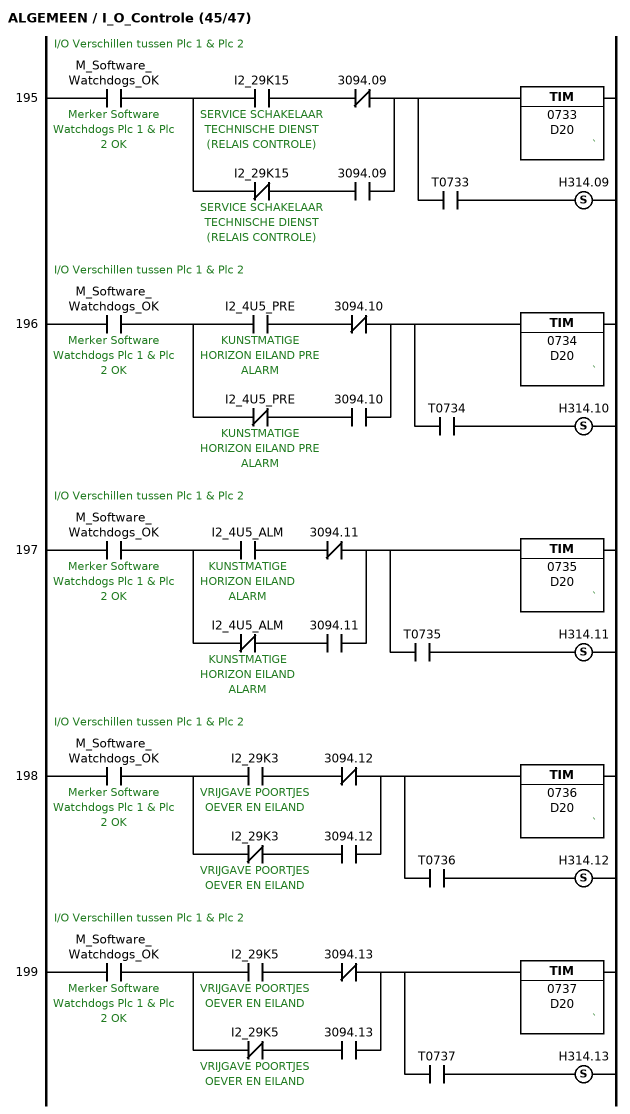
; [picture p253: ALGEMEEN / I_O_Controle, rungs 195-199]
; rung 195: I/O Verschillen tussen Plc 1 & Plc 2
LD M_Software_Watchdogs_OK  ; Merker Software Watchdogs Plc 1 & Plc 2 OK
LD I2_29K15  ; SERVICE SCHAKELAAR TECHNISCHE DIENST (RELAIS CONTROLE)
ANDNOT 3094.09
LDNOT I2_29K15  ; SERVICE SCHAKELAAR TECHNISCHE DIENST (RELAIS CONTROLE)
AND 3094.09
ORLD
ANDLD
TIM 0733 D20  ; `
AND T0733
SET H314.09
; rung 196: I/O Verschillen tussen Plc 1 & Plc 2
LD M_Software_Watchdogs_OK  ; Merker Software Watchdogs Plc 1 & Plc 2 OK
LD I2_4U5_PRE  ; KUNSTMATIGE HORIZON EILAND PRE ALARM
ANDNOT 3094.10
LDNOT I2_4U5_PRE  ; KUNSTMATIGE HORIZON EILAND PRE ALARM
AND 3094.10
ORLD
ANDLD
TIM 0734 D20  ; `
AND T0734
SET H314.10
; rung 197: I/O Verschillen tussen Plc 1 & Plc 2
LD M_Software_Watchdogs_OK  ; Merker Software Watchdogs Plc 1 & Plc 2 OK
LD I2_4U5_ALM  ; KUNSTMATIGE HORIZON EILAND ALARM
ANDNOT 3094.11
LDNOT I2_4U5_ALM  ; KUNSTMATIGE HORIZON EILAND ALARM
AND 3094.11
ORLD
ANDLD
TIM 0735 D20  ; `
AND T0735
SET H314.11
; rung 198: I/O Verschillen tussen Plc 1 & Plc 2
LD M_Software_Watchdogs_OK  ; Merker Software Watchdogs Plc 1 & Plc 2 OK
LD I2_29K3  ; VRIJGAVE POORTJES OEVER EN EILAND
ANDNOT 3094.12
LDNOT I2_29K3  ; VRIJGAVE POORTJES OEVER EN EILAND
AND 3094.12
ORLD
ANDLD
TIM 0736 D20  ; `
AND T0736
SET H314.12
; rung 199: I/O Verschillen tussen Plc 1 & Plc 2
LD M_Software_Watchdogs_OK  ; Merker Software Watchdogs Plc 1 & Plc 2 OK
LD I2_29K5  ; VRIJGAVE POORTJES OEVER EN EILAND
ANDNOT 3094.13
LDNOT I2_29K5  ; VRIJGAVE POORTJES OEVER EN EILAND
AND 3094.13
ORLD
ANDLD
TIM 0737 D20  ; `
AND T0737
SET H314.13

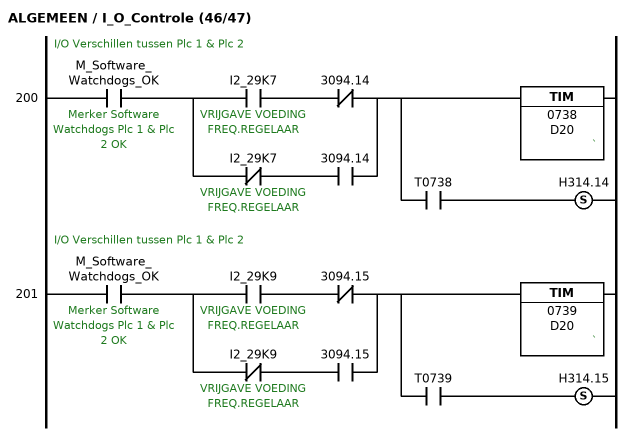
; rung 200: I/O Verschillen tussen Plc 1 & Plc 2
LD M_Software_Watchdogs_OK  ; Merker Software Watchdogs Plc 1 & Plc 2 OK
LD I2_29K7  ; VRIJGAVE VOEDING FREQ.REGELAAR
ANDNOT 3094.14
LDNOT I2_29K7  ; VRIJGAVE VOEDING FREQ.REGELAAR
AND 3094.14
ORLD
ANDLD
TIM 0738 D20  ; `
AND T0738
SET H314.14
; rung 201: I/O Verschillen tussen Plc 1 & Plc 2
LD M_Software_Watchdogs_OK  ; Merker Software Watchdogs Plc 1 & Plc 2 OK
LD I2_29K9  ; VRIJGAVE VOEDING FREQ.REGELAAR
ANDNOT 3094.15
LDNOT I2_29K9  ; VRIJGAVE VOEDING FREQ.REGELAAR
AND 3094.15
ORLD
ANDLD
TIM 0739 D20  ; `
AND T0739
SET H314.15

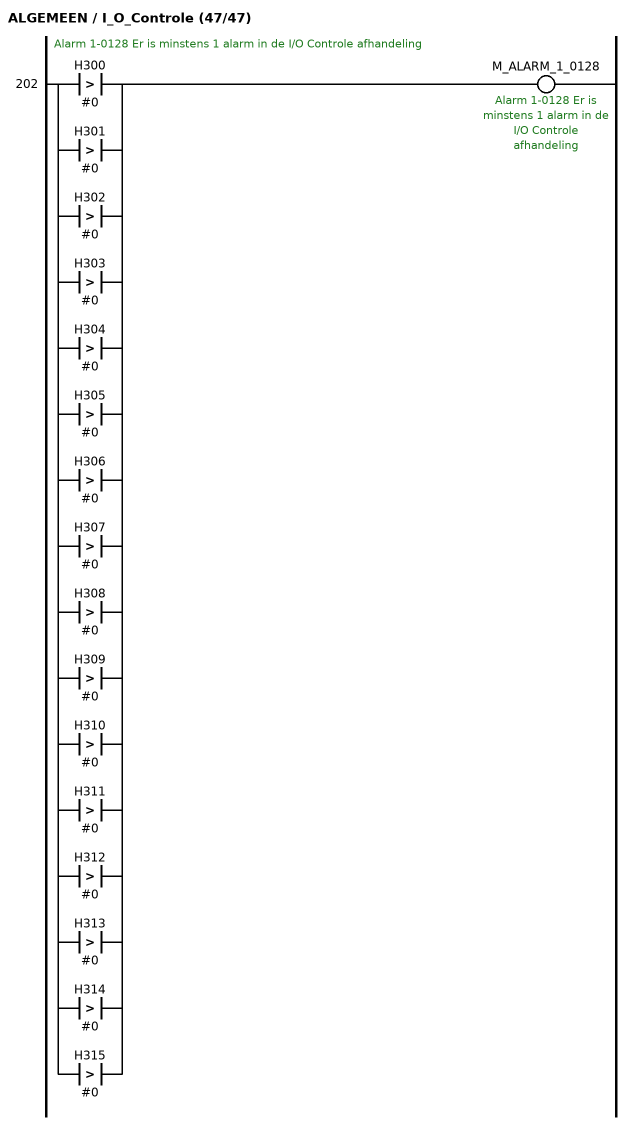
; rung 202: Alarm 1-0128 Er is minstens 1 alarm in de I/O Controle afhandeling
LD>(320) H300 #0
OR>(320) H301 #0
OR>(320) H302 #0
OR>(320) H303 #0
OR>(320) H304 #0
OR>(320) H305 #0
OR>(320) H306 #0
OR>(320) H307 #0
OR>(320) H308 #0
OR>(320) H309 #0
OR>(320) H310 #0
OR>(320) H311 #0
OR>(320) H312 #0
OR>(320) H313 #0
OR>(320) H314 #0
OR>(320) H315 #0
OUT M_ALARM_1_0128  ; Alarm 1-0128 Er is minstens 1 alarm in de I/O Controle afhandeling

### Section Voedingen

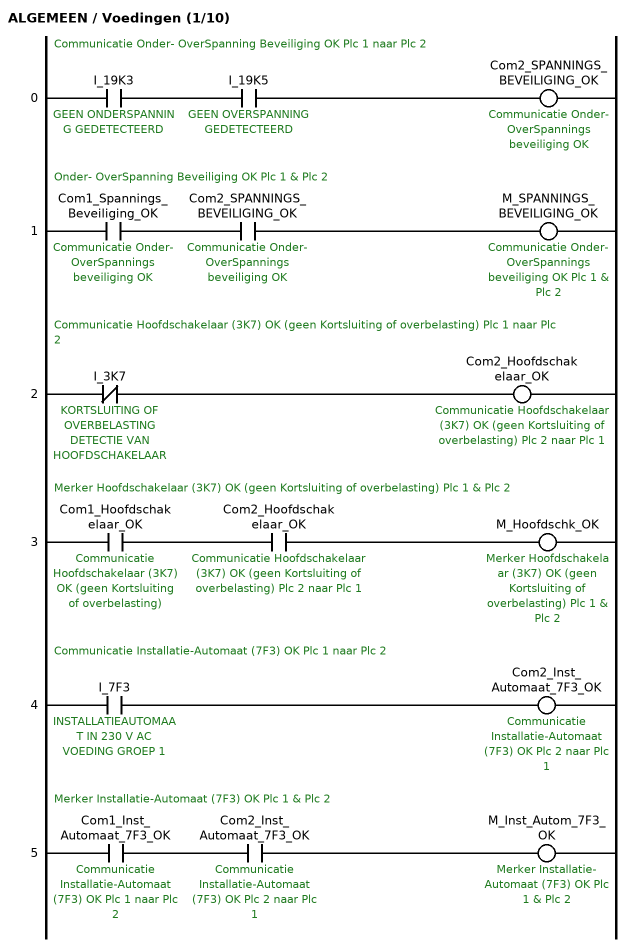
; rung 0: Communicatie Onder- OverSpanning Beveiliging OK Plc 1 naar Plc 2
LD I_19K3  ; GEEN ONDERSPANNING GEDETECTEERD
AND I_19K5  ; GEEN OVERSPANNING GEDETECTEERD
OUT Com2_SPANNINGS_BEVEILIGING_OK  ; Communicatie Onder- OverSpannings beveiliging OK
; rung 1: Onder- OverSpanning Beveiliging OK Plc 1 & Plc 2
LD Com1_Spannings_Beveiliging_OK  ; Communicatie Onder- OverSpannings beveiliging OK
AND Com2_SPANNINGS_BEVEILIGING_OK  ; Communicatie Onder- OverSpannings beveiliging OK
OUT M_SPANNINGS_BEVEILIGING_OK  ; Communicatie Onder- OverSpannings beveiliging OK Plc 1 & Plc 2
; rung 2: Communicatie Hoofdschakelaar (3K7) OK (geen Kortsluiting of overbelasting) Plc 1 naar Plc 2
LDNOT I_3K7  ; KORTSLUITING OF OVERBELASTING DETECTIE VAN HOOFDSCHAKELAAR
OUT Com2_Hoofdschakelaar_OK  ; Communicatie Hoofdschakelaar (3K7) OK (geen Kortsluiting of overbelasting) Plc 2 naar Plc 1
; rung 3: Merker Hoofdschakelaar (3K7) OK (geen Kortsluiting of overbelasting) Plc 1 & Plc 2
LD Com1_Hoofdschakelaar_OK  ; Communicatie Hoofdschakelaar (3K7) OK (geen Kortsluiting of overbelasting)
AND Com2_Hoofdschakelaar_OK  ; Communicatie Hoofdschakelaar (3K7) OK (geen Kortsluiting of overbelasting) Plc 2 naar Plc 1
OUT M_Hoofdschk_OK  ; Merker Hoofdschakelaar (3K7) OK (geen Kortsluiting of overbelasting) Plc 1 & Plc 2
; rung 4: Communicatie Installatie-Automaat (7F3) OK Plc 1 naar Plc 2
LD I_7F3  ; INSTALLATIEAUTOMAAT IN 230 V AC VOEDING GROEP 1
OUT Com2_Inst_Automaat_7F3_OK  ; Communicatie Installatie-Automaat (7F3) OK Plc 2 naar Plc 1
; rung 5: Merker Installatie-Automaat (7F3) OK Plc 1 & Plc 2
LD Com1_Inst_Automaat_7F3_OK  ; Communicatie Installatie-Automaat (7F3) OK Plc 1 naar Plc 2
AND Com2_Inst_Automaat_7F3_OK  ; Communicatie Installatie-Automaat (7F3) OK Plc 2 naar Plc 1
OUT M_Inst_Autom_7F3_OK  ; Merker Installatie-Automaat (7F3) OK Plc 1 & Plc 2

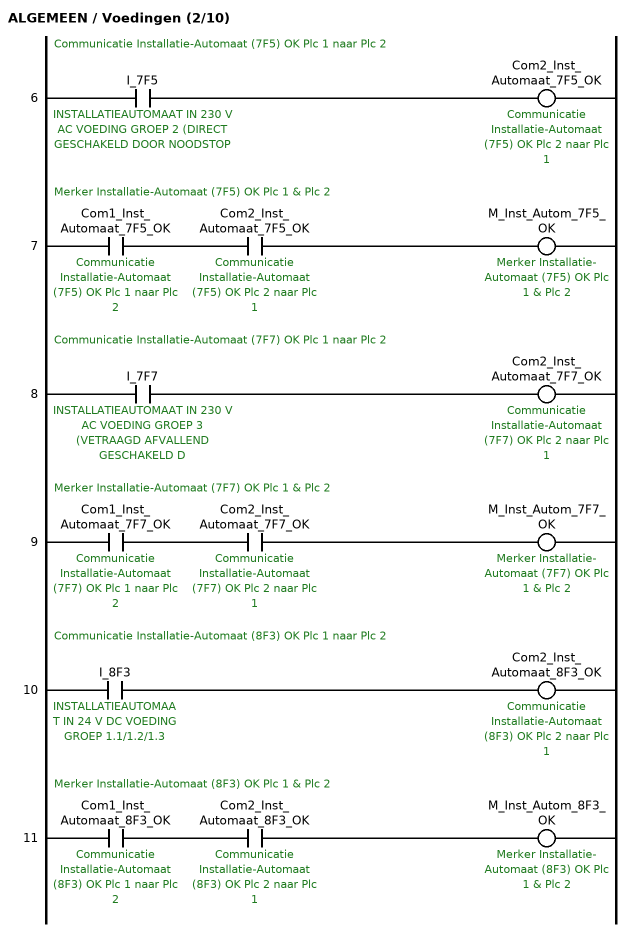
; rung 6: Communicatie Installatie-Automaat (7F5) OK Plc 1 naar Plc 2
LD I_7F5  ; INSTALLATIEAUTOMAAT IN 230 V AC VOEDING GROEP 2 (DIRECT GESCHAKELD DOOR NOODSTOP
OUT Com2_Inst_Automaat_7F5_OK  ; Communicatie Installatie-Automaat (7F5) OK Plc 2 naar Plc 1
; rung 7: Merker Installatie-Automaat (7F5) OK Plc 1 & Plc 2
LD Com1_Inst_Automaat_7F5_OK  ; Communicatie Installatie-Automaat (7F5) OK Plc 1 naar Plc 2
AND Com2_Inst_Automaat_7F5_OK  ; Communicatie Installatie-Automaat (7F5) OK Plc 2 naar Plc 1
OUT M_Inst_Autom_7F5_OK  ; Merker Installatie-Automaat (7F5) OK Plc 1 & Plc 2
; rung 8: Communicatie Installatie-Automaat (7F7) OK Plc 1 naar Plc 2
LD I_7F7  ; INSTALLATIEAUTOMAAT IN 230 V AC VOEDING GROEP 3 (VETRAAGD AFVALLEND GESCHAKELD D
OUT Com2_Inst_Automaat_7F7_OK  ; Communicatie Installatie-Automaat (7F7) OK Plc 2 naar Plc 1
; rung 9: Merker Installatie-Automaat (7F7) OK Plc 1 & Plc 2
LD Com1_Inst_Automaat_7F7_OK  ; Communicatie Installatie-Automaat (7F7) OK Plc 1 naar Plc 2
AND Com2_Inst_Automaat_7F7_OK  ; Communicatie Installatie-Automaat (7F7) OK Plc 2 naar Plc 1
OUT M_Inst_Autom_7F7_OK  ; Merker Installatie-Automaat (7F7) OK Plc 1 & Plc 2
; rung 10: Communicatie Installatie-Automaat (8F3) OK Plc 1 naar Plc 2
LD I_8F3  ; INSTALLATIEAUTOMAAT IN 24 V DC VOEDING GROEP 1.1/1.2/1.3
OUT Com2_Inst_Automaat_8F3_OK  ; Communicatie Installatie-Automaat (8F3) OK Plc 2 naar Plc 1
; rung 11: Merker Installatie-Automaat (8F3) OK Plc 1 & Plc 2
LD Com1_Inst_Automaat_8F3_OK  ; Communicatie Installatie-Automaat (8F3) OK Plc 1 naar Plc 2
AND Com2_Inst_Automaat_8F3_OK  ; Communicatie Installatie-Automaat (8F3) OK Plc 2 naar Plc 1
OUT M_Inst_Autom_8F3_OK  ; Merker Installatie-Automaat (8F3) OK Plc 1 & Plc 2

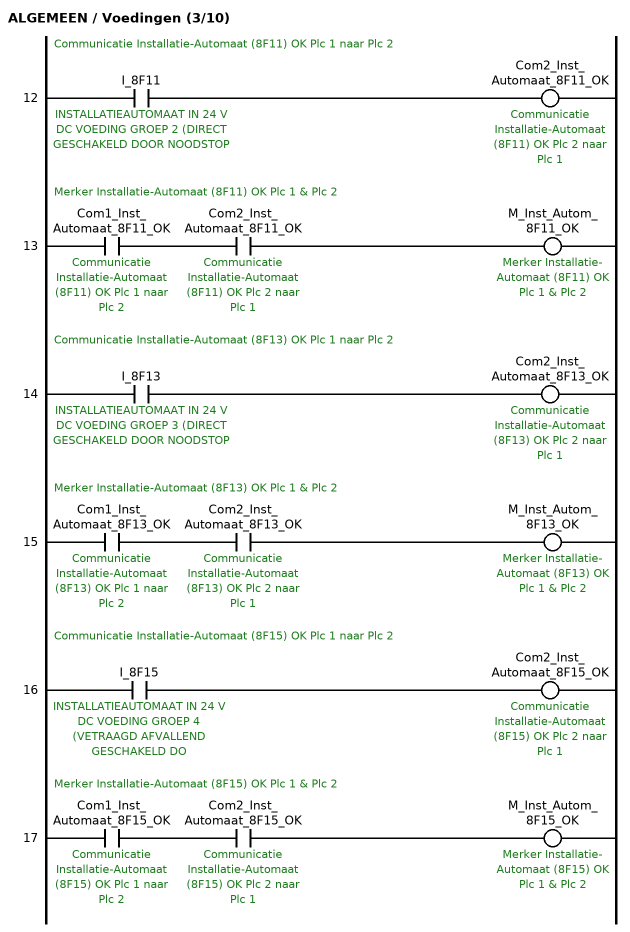
; rung 12: Communicatie Installatie-Automaat (8F11) OK Plc 1 naar Plc 2
LD I_8F11  ; INSTALLATIEAUTOMAAT IN 24 V DC VOEDING GROEP 2 (DIRECT GESCHAKELD DOOR NOODSTOP
OUT Com2_Inst_Automaat_8F11_OK  ; Communicatie Installatie-Automaat (8F11) OK Plc 2 naar Plc 1
; rung 13: Merker Installatie-Automaat (8F11) OK Plc 1 & Plc 2
LD Com1_Inst_Automaat_8F11_OK  ; Communicatie Installatie-Automaat (8F11) OK Plc 1 naar Plc 2
AND Com2_Inst_Automaat_8F11_OK  ; Communicatie Installatie-Automaat (8F11) OK Plc 2 naar Plc 1
OUT M_Inst_Autom_8F11_OK  ; Merker Installatie-Automaat (8F11) OK Plc 1 & Plc 2
; rung 14: Communicatie Installatie-Automaat (8F13) OK Plc 1 naar Plc 2
LD I_8F13  ; INSTALLATIEAUTOMAAT IN 24 V DC VOEDING GROEP 3 (DIRECT GESCHAKELD DOOR NOODSTOP
OUT Com2_Inst_Automaat_8F13_OK  ; Communicatie Installatie-Automaat (8F13) OK Plc 2 naar Plc 1
; rung 15: Merker Installatie-Automaat (8F13) OK Plc 1 & Plc 2
LD Com1_Inst_Automaat_8F13_OK  ; Communicatie Installatie-Automaat (8F13) OK Plc 1 naar Plc 2
AND Com2_Inst_Automaat_8F13_OK  ; Communicatie Installatie-Automaat (8F13) OK Plc 2 naar Plc 1
OUT M_Inst_Autom_8F13_OK  ; Merker Installatie-Automaat (8F13) OK Plc 1 & Plc 2
; rung 16: Communicatie Installatie-Automaat (8F15) OK Plc 1 naar Plc 2
LD I_8F15  ; INSTALLATIEAUTOMAAT IN 24 V DC VOEDING GROEP 4 (VETRAAGD AFVALLEND GESCHAKELD DO
OUT Com2_Inst_Automaat_8F15_OK  ; Communicatie Installatie-Automaat (8F15) OK Plc 2 naar Plc 1
; rung 17: Merker Installatie-Automaat (8F15) OK Plc 1 & Plc 2
LD Com1_Inst_Automaat_8F15_OK  ; Communicatie Installatie-Automaat (8F15) OK Plc 1 naar Plc 2
AND Com2_Inst_Automaat_8F15_OK  ; Communicatie Installatie-Automaat (8F15) OK Plc 2 naar Plc 1
OUT M_Inst_Autom_8F15_OK  ; Merker Installatie-Automaat (8F15) OK Plc 1 & Plc 2

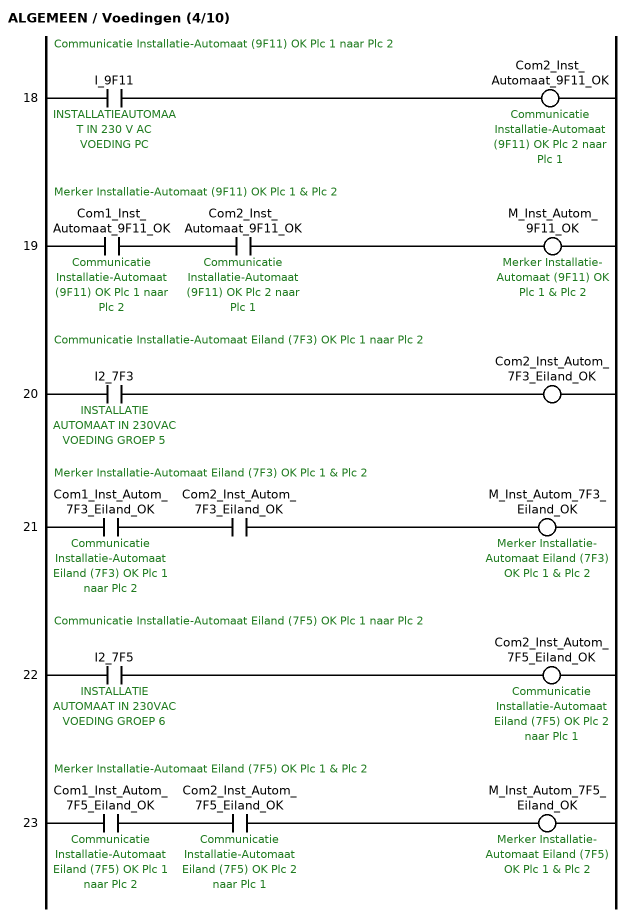
; rung 18: Communicatie Installatie-Automaat (9F11) OK Plc 1 naar Plc 2
LD I_9F11  ; INSTALLATIEAUTOMAAT IN 230 V AC VOEDING PC
OUT Com2_Inst_Automaat_9F11_OK  ; Communicatie Installatie-Automaat (9F11) OK Plc 2 naar Plc 1
; rung 19: Merker Installatie-Automaat (9F11) OK Plc 1 & Plc 2
LD Com1_Inst_Automaat_9F11_OK  ; Communicatie Installatie-Automaat (9F11) OK Plc 1 naar Plc 2
AND Com2_Inst_Automaat_9F11_OK  ; Communicatie Installatie-Automaat (9F11) OK Plc 2 naar Plc 1
OUT M_Inst_Autom_9F11_OK  ; Merker Installatie-Automaat (9F11) OK Plc 1 & Plc 2
; rung 20: Communicatie Installatie-Automaat Eiland (7F3) OK Plc 1 naar Plc 2
LD I2_7F3  ; INSTALLATIE AUTOMAAT IN 230VAC VOEDING GROEP 5
OUT Com2_Inst_Autom_7F3_Eiland_OK
; rung 21: Merker Installatie-Automaat Eiland (7F3) OK Plc 1 & Plc 2
LD Com1_Inst_Autom_7F3_Eiland_OK  ; Communicatie Installatie-Automaat Eiland (7F3) OK Plc 1 naar Plc 2
AND Com2_Inst_Autom_7F3_Eiland_OK
OUT M_Inst_Autom_7F3_Eiland_OK  ; Merker Installatie-Automaat Eiland (7F3) OK Plc 1 & Plc 2
; rung 22: Communicatie Installatie-Automaat Eiland (7F5) OK Plc 1 naar Plc 2
LD I2_7F5  ; INSTALLATIE AUTOMAAT IN 230VAC VOEDING GROEP 6
OUT Com2_Inst_Autom_7F5_Eiland_OK  ; Communicatie Installatie-Automaat Eiland (7F5) OK Plc 2 naar Plc 1
; rung 23: Merker Installatie-Automaat Eiland (7F5) OK Plc 1 & Plc 2
LD Com1_Inst_Autom_7F5_Eiland_OK  ; Communicatie Installatie-Automaat Eiland (7F5) OK Plc 1 naar Plc 2
AND Com2_Inst_Autom_7F5_Eiland_OK  ; Communicatie Installatie-Automaat Eiland (7F5) OK Plc 2 naar Plc 1
OUT M_Inst_Autom_7F5_Eiland_OK  ; Merker Installatie-Automaat Eiland (7F5) OK Plc 1 & Plc 2

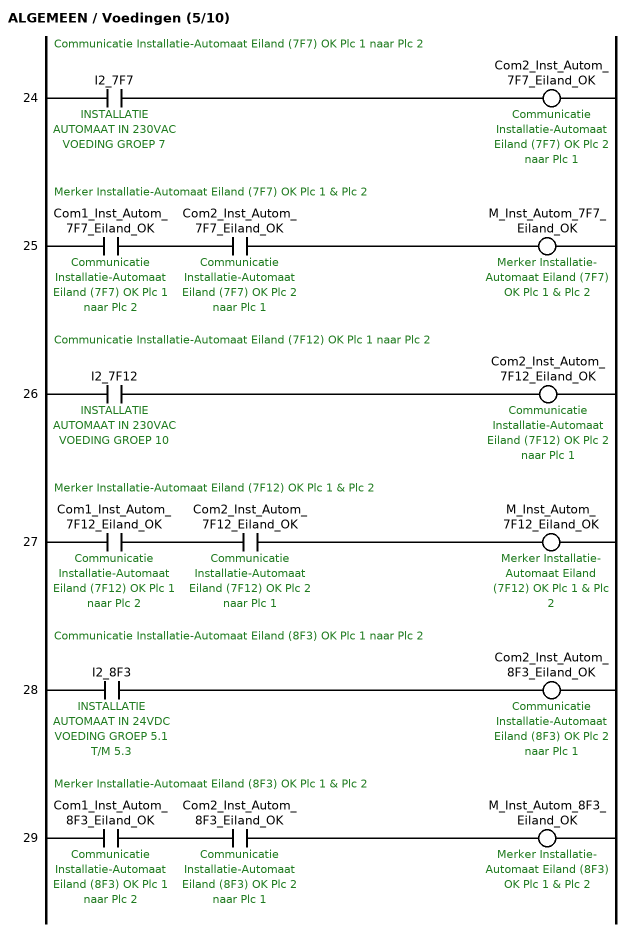
; rung 24: Communicatie Installatie-Automaat Eiland (7F7) OK Plc 1 naar Plc 2
LD I2_7F7  ; INSTALLATIE AUTOMAAT IN 230VAC VOEDING GROEP 7
OUT Com2_Inst_Autom_7F7_Eiland_OK  ; Communicatie Installatie-Automaat Eiland (7F7) OK Plc 2 naar Plc 1
; rung 25: Merker Installatie-Automaat Eiland (7F7) OK Plc 1 & Plc 2
LD Com1_Inst_Autom_7F7_Eiland_OK  ; Communicatie Installatie-Automaat Eiland (7F7) OK Plc 1 naar Plc 2
AND Com2_Inst_Autom_7F7_Eiland_OK  ; Communicatie Installatie-Automaat Eiland (7F7) OK Plc 2 naar Plc 1
OUT M_Inst_Autom_7F7_Eiland_OK  ; Merker Installatie-Automaat Eiland (7F7) OK Plc 1 & Plc 2
; rung 26: Communicatie Installatie-Automaat Eiland (7F12) OK Plc 1 naar Plc 2
LD I2_7F12  ; INSTALLATIE AUTOMAAT IN 230VAC VOEDING GROEP 10
OUT Com2_Inst_Autom_7F12_Eiland_OK  ; Communicatie Installatie-Automaat Eiland (7F12) OK Plc 2 naar Plc 1
; rung 27: Merker Installatie-Automaat Eiland (7F12) OK Plc 1 & Plc 2
LD Com1_Inst_Autom_7F12_Eiland_OK  ; Communicatie Installatie-Automaat Eiland (7F12) OK Plc 1 naar Plc 2
AND Com2_Inst_Autom_7F12_Eiland_OK  ; Communicatie Installatie-Automaat Eiland (7F12) OK Plc 2 naar Plc 1
OUT M_Inst_Autom_7F12_Eiland_OK  ; Merker Installatie-Automaat Eiland (7F12) OK Plc 1 & Plc 2
; rung 28: Communicatie Installatie-Automaat Eiland (8F3) OK Plc 1 naar Plc 2
LD I2_8F3  ; INSTALLATIE AUTOMAAT IN 24VDC VOEDING GROEP 5.1 T/M 5.3
OUT Com2_Inst_Autom_8F3_Eiland_OK  ; Communicatie Installatie-Automaat Eiland (8F3) OK Plc 2 naar Plc 1
; rung 29: Merker Installatie-Automaat Eiland (8F3) OK Plc 1 & Plc 2
LD Com1_Inst_Autom_8F3_Eiland_OK  ; Communicatie Installatie-Automaat Eiland (8F3) OK Plc 1 naar Plc 2
AND Com2_Inst_Autom_8F3_Eiland_OK  ; Communicatie Installatie-Automaat Eiland (8F3) OK Plc 2 naar Plc 1
OUT M_Inst_Autom_8F3_Eiland_OK  ; Merker Installatie-Automaat Eiland (8F3) OK Plc 1 & Plc 2

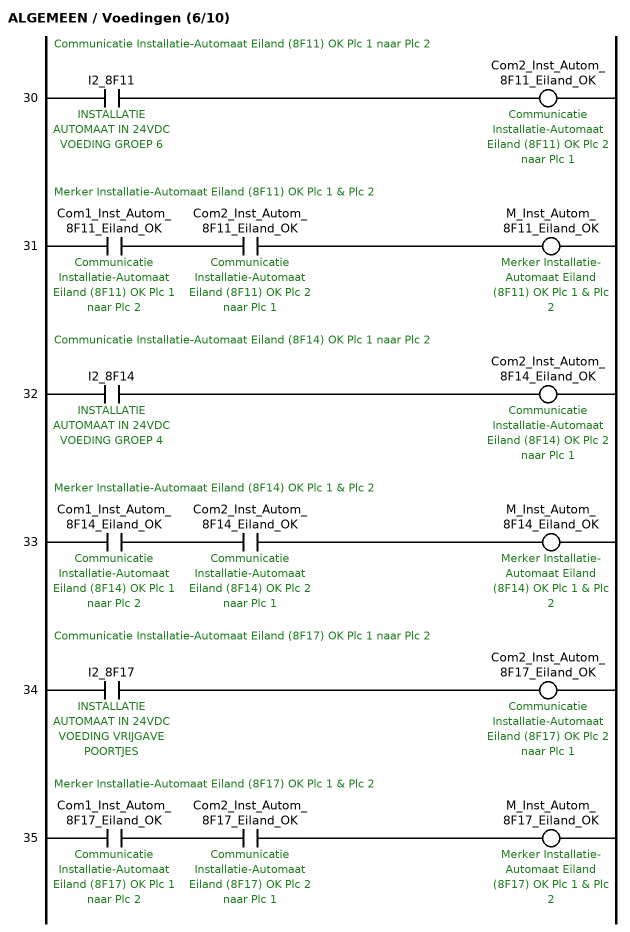
; rung 30: Communicatie Installatie-Automaat Eiland (8F11) OK Plc 1 naar Plc 2
LD I2_8F11  ; INSTALLATIE AUTOMAAT IN 24VDC VOEDING GROEP 6
OUT Com2_Inst_Autom_8F11_Eiland_OK  ; Communicatie Installatie-Automaat Eiland (8F11) OK Plc 2 naar Plc 1
; rung 31: Merker Installatie-Automaat Eiland (8F11) OK Plc 1 & Plc 2
LD Com1_Inst_Autom_8F11_Eiland_OK  ; Communicatie Installatie-Automaat Eiland (8F11) OK Plc 1 naar Plc 2
AND Com2_Inst_Autom_8F11_Eiland_OK  ; Communicatie Installatie-Automaat Eiland (8F11) OK Plc 2 naar Plc 1
OUT M_Inst_Autom_8F11_Eiland_OK  ; Merker Installatie-Automaat Eiland (8F11) OK Plc 1 & Plc 2
; rung 32: Communicatie Installatie-Automaat Eiland (8F14) OK Plc 1 naar Plc 2
LD I2_8F14  ; INSTALLATIE AUTOMAAT IN 24VDC VOEDING GROEP 4
OUT Com2_Inst_Autom_8F14_Eiland_OK  ; Communicatie Installatie-Automaat Eiland (8F14) OK Plc 2 naar Plc 1
; rung 33: Merker Installatie-Automaat Eiland (8F14) OK Plc 1 & Plc 2
LD Com1_Inst_Autom_8F14_Eiland_OK  ; Communicatie Installatie-Automaat Eiland (8F14) OK Plc 1 naar Plc 2
AND Com2_Inst_Autom_8F14_Eiland_OK  ; Communicatie Installatie-Automaat Eiland (8F14) OK Plc 2 naar Plc 1
OUT M_Inst_Autom_8F14_Eiland_OK  ; Merker Installatie-Automaat Eiland (8F14) OK Plc 1 & Plc 2
; rung 34: Communicatie Installatie-Automaat Eiland (8F17) OK Plc 1 naar Plc 2
LD I2_8F17  ; INSTALLATIE AUTOMAAT IN 24VDC VOEDING VRIJGAVE POORTJES
OUT Com2_Inst_Autom_8F17_Eiland_OK  ; Communicatie Installatie-Automaat Eiland (8F17) OK Plc 2 naar Plc 1
; rung 35: Merker Installatie-Automaat Eiland (8F17) OK Plc 1 & Plc 2
LD Com1_Inst_Autom_8F17_Eiland_OK  ; Communicatie Installatie-Automaat Eiland (8F17) OK Plc 1 naar Plc 2
AND Com2_Inst_Autom_8F17_Eiland_OK  ; Communicatie Installatie-Automaat Eiland (8F17) OK Plc 2 naar Plc 1
OUT M_Inst_Autom_8F17_Eiland_OK  ; Merker Installatie-Automaat Eiland (8F17) OK Plc 1 & Plc 2

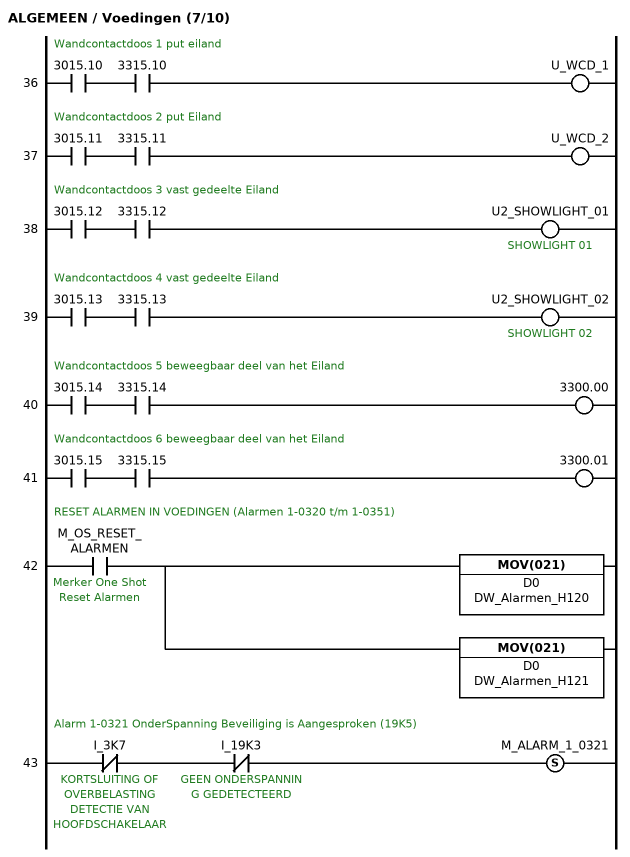
; rung 36: Wandcontactdoos 1 put eiland
LD 3015.10
AND 3315.10
OUT U_WCD_1
; rung 37: Wandcontactdoos 2 put Eiland
LD 3015.11
AND 3315.11
OUT U_WCD_2
; rung 38: Wandcontactdoos 3 vast gedeelte Eiland
LD 3015.12
AND 3315.12
OUT U2_SHOWLIGHT_01  ; SHOWLIGHT 01
; rung 39: Wandcontactdoos 4 vast gedeelte Eiland
LD 3015.13
AND 3315.13
OUT U2_SHOWLIGHT_02  ; SHOWLIGHT 02
; rung 40: Wandcontactdoos 5 beweegbaar deel van het Eiland
LD 3015.14
AND 3315.14
OUT 3300.00
; rung 41: Wandcontactdoos 6 beweegbaar deel van het Eiland
LD 3015.15
AND 3315.15
OUT 3300.01
; rung 42: RESET ALARMEN IN VOEDINGEN (Alarmen 1-0320 t/m 1-0351)
LD M_OS_RESET_ALARMEN  ; Merker One Shot Reset Alarmen
MOV(021) D0 DW_Alarmen_H120
MOV(021) D0 DW_Alarmen_H121
; rung 43: Alarm 1-0321 OnderSpanning Beveiliging is Aangesproken (19K5)
LDNOT I_3K7  ; KORTSLUITING OF OVERBELASTING DETECTIE VAN HOOFDSCHAKELAAR
ANDNOT I_19K3  ; GEEN ONDERSPANNING GEDETECTEERD
SET M_ALARM_1_0321

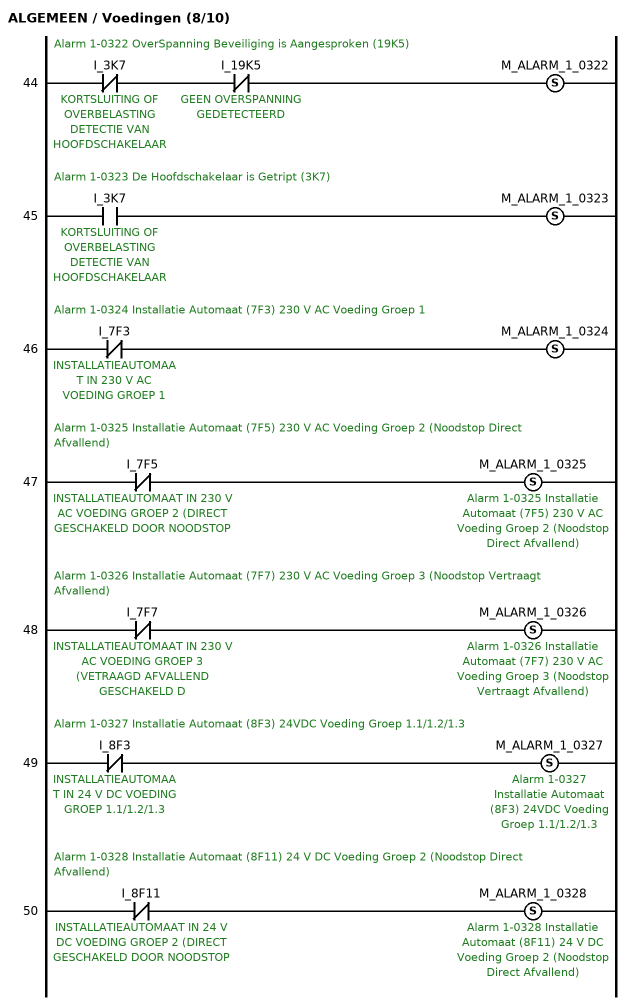
; rung 44: Alarm 1-0322 OverSpanning Beveiliging is Aangesproken (19K5)
LDNOT I_3K7  ; KORTSLUITING OF OVERBELASTING DETECTIE VAN HOOFDSCHAKELAAR
ANDNOT I_19K5  ; GEEN OVERSPANNING GEDETECTEERD
SET M_ALARM_1_0322
; rung 45: Alarm 1-0323 De Hoofdschakelaar is Getript (3K7)
LD I_3K7  ; KORTSLUITING OF OVERBELASTING DETECTIE VAN HOOFDSCHAKELAAR
SET M_ALARM_1_0323
; rung 46: Alarm 1-0324 Installatie Automaat (7F3) 230 V AC Voeding Groep 1
LDNOT I_7F3  ; INSTALLATIEAUTOMAAT IN 230 V AC VOEDING GROEP 1
SET M_ALARM_1_0324
; rung 47: Alarm 1-0325 Installatie Automaat (7F5) 230 V AC Voeding Groep 2 (Noodstop Direct Afvallend)
LDNOT I_7F5  ; INSTALLATIEAUTOMAAT IN 230 V AC VOEDING GROEP 2 (DIRECT GESCHAKELD DOOR NOODSTOP
SET M_ALARM_1_0325  ; Alarm 1-0325 Installatie Automaat (7F5) 230 V AC Voeding Groep 2 (Noodstop Direct Afvallend)
; rung 48: Alarm 1-0326 Installatie Automaat (7F7) 230 V AC Voeding Groep 3 (Noodstop Vertraagt Afvallend)
LDNOT I_7F7  ; INSTALLATIEAUTOMAAT IN 230 V AC VOEDING GROEP 3 (VETRAAGD AFVALLEND GESCHAKELD D
SET M_ALARM_1_0326  ; Alarm 1-0326 Installatie Automaat (7F7) 230 V AC Voeding Groep 3 (Noodstop Vertraagt Afvallend)
; rung 49: Alarm 1-0327 Installatie Automaat (8F3) 24VDC Voeding Groep 1.1/1.2/1.3
LDNOT I_8F3  ; INSTALLATIEAUTOMAAT IN 24 V DC VOEDING GROEP 1.1/1.2/1.3
SET M_ALARM_1_0327  ; Alarm 1-0327 Installatie Automaat (8F3) 24VDC Voeding Groep 1.1/1.2/1.3
; rung 50: Alarm 1-0328 Installatie Automaat (8F11) 24 V DC Voeding Groep 2 (Noodstop Direct Afvallend)
LDNOT I_8F11  ; INSTALLATIEAUTOMAAT IN 24 V DC VOEDING GROEP 2 (DIRECT GESCHAKELD DOOR NOODSTOP
SET M_ALARM_1_0328  ; Alarm 1-0328 Installatie Automaat (8F11) 24 V DC Voeding Groep 2 (Noodstop Direct Afvallend)

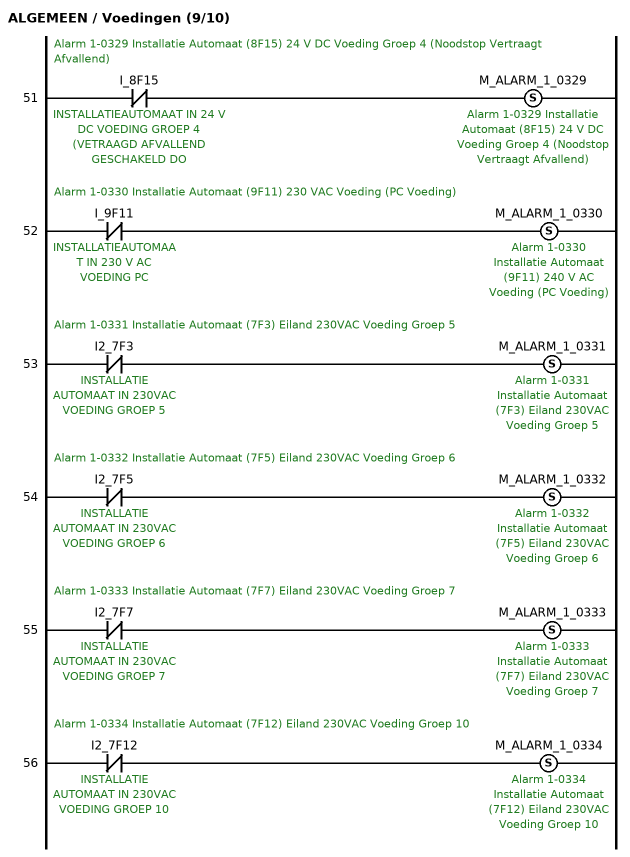
; rung 51: Alarm 1-0329 Installatie Automaat (8F15) 24 V DC Voeding Groep 4 (Noodstop Vertraagt Afvallend)
LDNOT I_8F15  ; INSTALLATIEAUTOMAAT IN 24 V DC VOEDING GROEP 4 (VETRAAGD AFVALLEND GESCHAKELD DO
SET M_ALARM_1_0329  ; Alarm 1-0329 Installatie Automaat (8F15) 24 V DC Voeding Groep 4 (Noodstop Vertraagt Afvallend)
; rung 52: Alarm 1-0330 Installatie Automaat (9F11) 230 VAC Voeding (PC Voeding)
LDNOT I_9F11  ; INSTALLATIEAUTOMAAT IN 230 V AC VOEDING PC
SET M_ALARM_1_0330  ; Alarm 1-0330 Installatie Automaat (9F11) 240 V AC Voeding (PC Voeding)
; rung 53: Alarm 1-0331 Installatie Automaat (7F3) Eiland 230VAC Voeding Groep 5
LDNOT I2_7F3  ; INSTALLATIE AUTOMAAT IN 230VAC VOEDING GROEP 5
SET M_ALARM_1_0331  ; Alarm 1-0331 Installatie Automaat (7F3) Eiland 230VAC Voeding Groep 5
; rung 54: Alarm 1-0332 Installatie Automaat (7F5) Eiland 230VAC Voeding Groep 6
LDNOT I2_7F5  ; INSTALLATIE AUTOMAAT IN 230VAC VOEDING GROEP 6
SET M_ALARM_1_0332  ; Alarm 1-0332 Installatie Automaat (7F5) Eiland 230VAC Voeding Groep 6
; rung 55: Alarm 1-0333 Installatie Automaat (7F7) Eiland 230VAC Voeding Groep 7
LDNOT I2_7F7  ; INSTALLATIE AUTOMAAT IN 230VAC VOEDING GROEP 7
SET M_ALARM_1_0333  ; Alarm 1-0333 Installatie Automaat (7F7) Eiland 230VAC Voeding Groep 7
; rung 56: Alarm 1-0334 Installatie Automaat (7F12) Eiland 230VAC Voeding Groep 10
LDNOT I2_7F12  ; INSTALLATIE AUTOMAAT IN 230VAC VOEDING GROEP 10
SET M_ALARM_1_0334  ; Alarm 1-0334 Installatie Automaat (7F12) Eiland 230VAC Voeding Groep 10

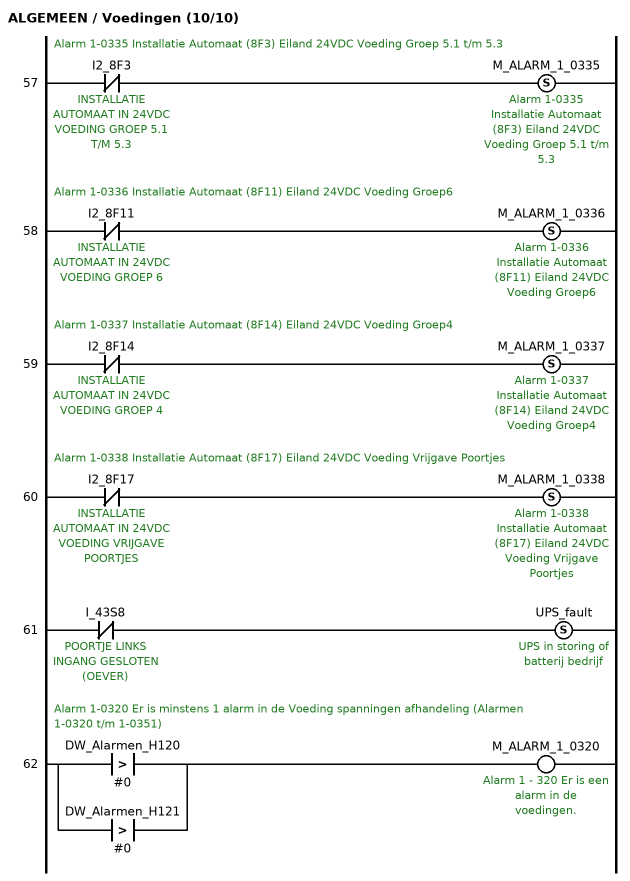
; rung 57: Alarm 1-0335 Installatie Automaat (8F3) Eiland 24VDC Voeding Groep 5.1 t/m 5.3
LDNOT I2_8F3  ; INSTALLATIE AUTOMAAT IN 24VDC VOEDING GROEP 5.1 T/M 5.3
SET M_ALARM_1_0335  ; Alarm 1-0335 Installatie Automaat (8F3) Eiland 24VDC Voeding Groep 5.1 t/m 5.3
; rung 58: Alarm 1-0336 Installatie Automaat (8F11) Eiland 24VDC Voeding Groep6
LDNOT I2_8F11  ; INSTALLATIE AUTOMAAT IN 24VDC VOEDING GROEP 6
SET M_ALARM_1_0336  ; Alarm 1-0336 Installatie Automaat (8F11) Eiland 24VDC Voeding Groep6
; rung 59: Alarm 1-0337 Installatie Automaat (8F14) Eiland 24VDC Voeding Groep4
LDNOT I2_8F14  ; INSTALLATIE AUTOMAAT IN 24VDC VOEDING GROEP 4
SET M_ALARM_1_0337  ; Alarm 1-0337 Installatie Automaat (8F14) Eiland 24VDC Voeding Groep4
; rung 60: Alarm 1-0338 Installatie Automaat (8F17) Eiland 24VDC Voeding Vrijgave Poortjes
LDNOT I2_8F17  ; INSTALLATIE AUTOMAAT IN 24VDC VOEDING VRIJGAVE POORTJES
SET M_ALARM_1_0338  ; Alarm 1-0338 Installatie Automaat (8F17) Eiland 24VDC Voeding Vrijgave Poortjes
; rung 61
LDNOT I_43S8  ; POORTJE LINKS INGANG GESLOTEN (OEVER)
SET UPS_fault  ; UPS in storing of batterij bedrijf
; rung 62: Alarm 1-0320 Er is minstens 1 alarm in de Voeding spanningen afhandeling (Alarmen 1-0320 t/m 1-0351)
LD>(320) DW_Alarmen_H120 #0
OR>(320) DW_Alarmen_H121 #0
OUT M_ALARM_1_0320  ; Alarm 1 - 320 Er is een alarm in de voedingen.

### Section Watch_Dog

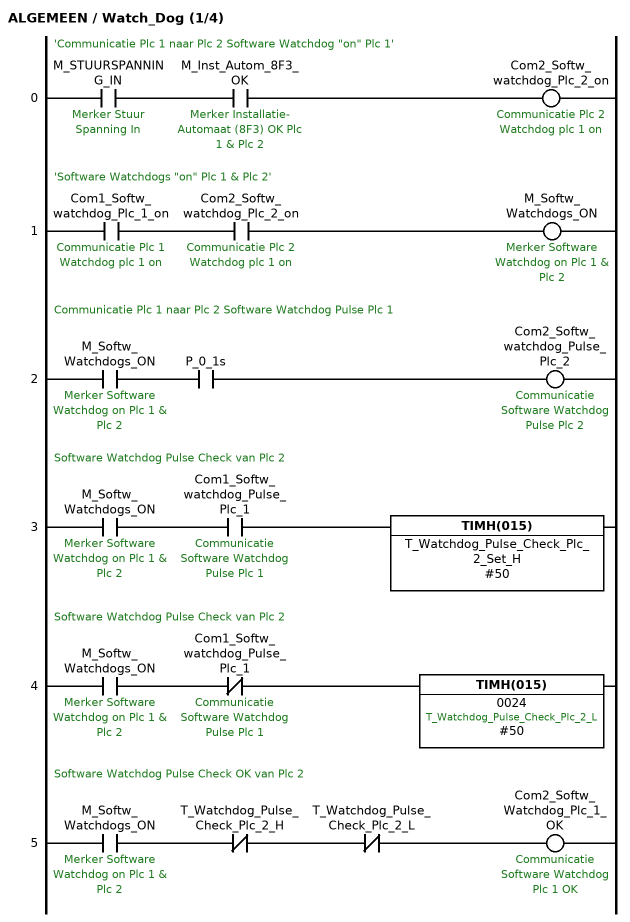
; rung 0: 'Communicatie Plc 1 naar Plc 2 Software Watchdog "on" Plc 1'
LD M_STUURSPANNING_IN  ; Merker Stuur Spanning In
AND M_Inst_Autom_8F3_OK  ; Merker Installatie-Automaat (8F3) OK Plc 1 & Plc 2
OUT Com2_Softw_watchdog_Plc_2_on  ; Communicatie Plc 2 Watchdog plc 1 on
; rung 1: 'Software Watchdogs "on" Plc 1 & Plc 2'
LD Com1_Softw_watchdog_Plc_1_on  ; Communicatie Plc 1 Watchdog plc 1 on
AND Com2_Softw_watchdog_Plc_2_on  ; Communicatie Plc 2 Watchdog plc 1 on
OUT M_Softw_Watchdogs_ON  ; Merker Software Watchdog on Plc 1 & Plc 2
; rung 2: Communicatie Plc 1 naar Plc 2 Software Watchdog Pulse Plc 1
LD M_Softw_Watchdogs_ON  ; Merker Software Watchdog on Plc 1 & Plc 2
AND P_0_1s
OUT Com2_Softw_watchdog_Pulse_Plc_2  ; Communicatie Software Watchdog Pulse Plc 2
; rung 3: Software Watchdog Pulse Check van Plc 2
LD M_Softw_Watchdogs_ON  ; Merker Software Watchdog on Plc 1 & Plc 2
AND Com1_Softw_watchdog_Pulse_Plc_1  ; Communicatie Software Watchdog Pulse Plc 1
TIMH(015) T_Watchdog_Pulse_Check_Plc_2_Set_H #50
; rung 4: Software Watchdog Pulse Check van Plc 2
LD M_Softw_Watchdogs_ON  ; Merker Software Watchdog on Plc 1 & Plc 2
ANDNOT Com1_Softw_watchdog_Pulse_Plc_1  ; Communicatie Software Watchdog Pulse Plc 1
TIMH(015) 0024 #50  ; T_Watchdog_Pulse_Check_Plc_2_L
; rung 5: Software Watchdog Pulse Check OK van Plc 2
LD M_Softw_Watchdogs_ON  ; Merker Software Watchdog on Plc 1 & Plc 2
ANDNOT T_Watchdog_Pulse_Check_Plc_2_H
ANDNOT T_Watchdog_Pulse_Check_Plc_2_L
OUT Com2_Softw_Watchdog_Plc_1_OK  ; Communicatie Software Watchdog Plc 1 OK

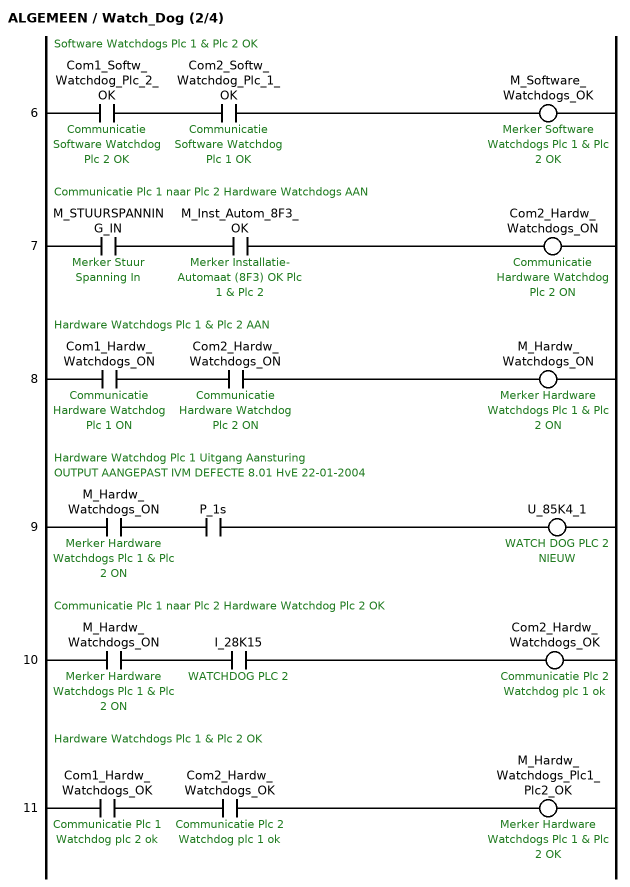
; rung 6: Software Watchdogs Plc 1 & Plc 2 OK
LD Com1_Softw_Watchdog_Plc_2_OK  ; Communicatie Software Watchdog Plc 2 OK
AND Com2_Softw_Watchdog_Plc_1_OK  ; Communicatie Software Watchdog Plc 1 OK
OUT M_Software_Watchdogs_OK  ; Merker Software Watchdogs Plc 1 & Plc 2 OK
; rung 7: Communicatie Plc 1 naar Plc 2 Hardware Watchdogs AAN
LD M_STUURSPANNING_IN  ; Merker Stuur Spanning In
AND M_Inst_Autom_8F3_OK  ; Merker Installatie-Automaat (8F3) OK Plc 1 & Plc 2
OUT Com2_Hardw_Watchdogs_ON  ; Communicatie Hardware Watchdog Plc 2 ON
; rung 8: Hardware Watchdogs Plc 1 & Plc 2 AAN
LD Com1_Hardw_Watchdogs_ON  ; Communicatie Hardware Watchdog Plc 1 ON
AND Com2_Hardw_Watchdogs_ON  ; Communicatie Hardware Watchdog Plc 2 ON
OUT M_Hardw_Watchdogs_ON  ; Merker Hardware Watchdogs Plc 1 & Plc 2 ON
; rung 9: Hardware Watchdog Plc 1 Uitgang Aansturing / OUTPUT AANGEPAST IVM DEFECTE 8.01 HvE 22-01-2004
LD M_Hardw_Watchdogs_ON  ; Merker Hardware Watchdogs Plc 1 & Plc 2 ON
AND P_1s
OUT U_85K4_1  ; WATCH DOG PLC 2 NIEUW
; rung 10: Communicatie Plc 1 naar Plc 2 Hardware Watchdog Plc 2 OK
LD M_Hardw_Watchdogs_ON  ; Merker Hardware Watchdogs Plc 1 & Plc 2 ON
AND I_28K15  ; WATCHDOG PLC 2
OUT Com2_Hardw_Watchdogs_OK  ; Communicatie Plc 2 Watchdog plc 1 ok
; rung 11: Hardware Watchdogs Plc 1 & Plc 2 OK
LD Com1_Hardw_Watchdogs_OK  ; Communicatie Plc 1 Watchdog plc 2 ok
AND Com2_Hardw_Watchdogs_OK  ; Communicatie Plc 2 Watchdog plc 1 ok
OUT M_Hardw_Watchdogs_Plc1_Plc2_OK  ; Merker Hardware Watchdogs Plc 1 & Plc 2 OK

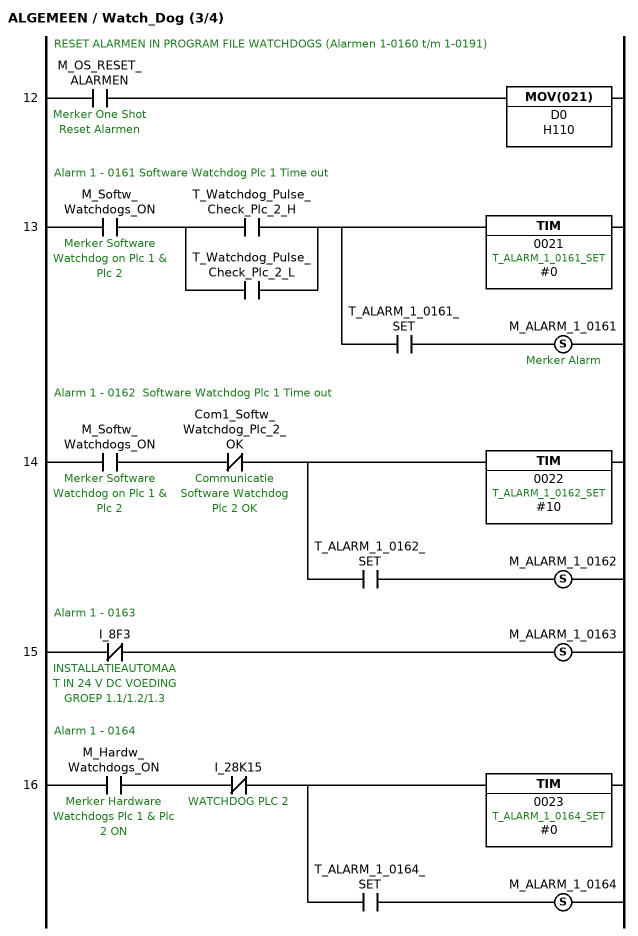
; rung 12: RESET ALARMEN IN PROGRAM FILE WATCHDOGS (Alarmen 1-0160 t/m 1-0191)
LD M_OS_RESET_ALARMEN  ; Merker One Shot Reset Alarmen
MOV(021) D0 H110
; rung 13: Alarm 1 - 0161 Software Watchdog Plc 1 Time out
LD M_Softw_Watchdogs_ON  ; Merker Software Watchdog on Plc 1 & Plc 2
LD T_Watchdog_Pulse_Check_Plc_2_H
OR T_Watchdog_Pulse_Check_Plc_2_L
ANDLD
TIM 0021 #0  ; T_ALARM_1_0161_SET
AND T_ALARM_1_0161_SET
SET M_ALARM_1_0161  ; Merker Alarm
; rung 14: Alarm 1 - 0162  Software Watchdog Plc 1 Time out
LD M_Softw_Watchdogs_ON  ; Merker Software Watchdog on Plc 1 & Plc 2
ANDNOT Com1_Softw_Watchdog_Plc_2_OK  ; Communicatie Software Watchdog Plc 2 OK
TIM 0022 #10  ; T_ALARM_1_0162_SET
AND T_ALARM_1_0162_SET
SET M_ALARM_1_0162
; rung 15: Alarm 1 - 0163
LDNOT I_8F3  ; INSTALLATIEAUTOMAAT IN 24 V DC VOEDING GROEP 1.1/1.2/1.3
SET M_ALARM_1_0163
; rung 16: Alarm 1 - 0164
LD M_Hardw_Watchdogs_ON  ; Merker Hardware Watchdogs Plc 1 & Plc 2 ON
ANDNOT I_28K15  ; WATCHDOG PLC 2
TIM 0023 #0  ; T_ALARM_1_0164_SET
AND T_ALARM_1_0164_SET
SET M_ALARM_1_0164

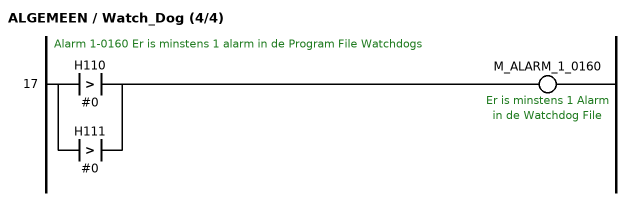
; rung 17: Alarm 1-0160 Er is minstens 1 alarm in de Program File Watchdogs
LD>(320) H110 #0
OR>(320) H111 #0
OUT M_ALARM_1_0160  ; Er is minstens 1 Alarm in de Watchdog File

### Section E_Stops

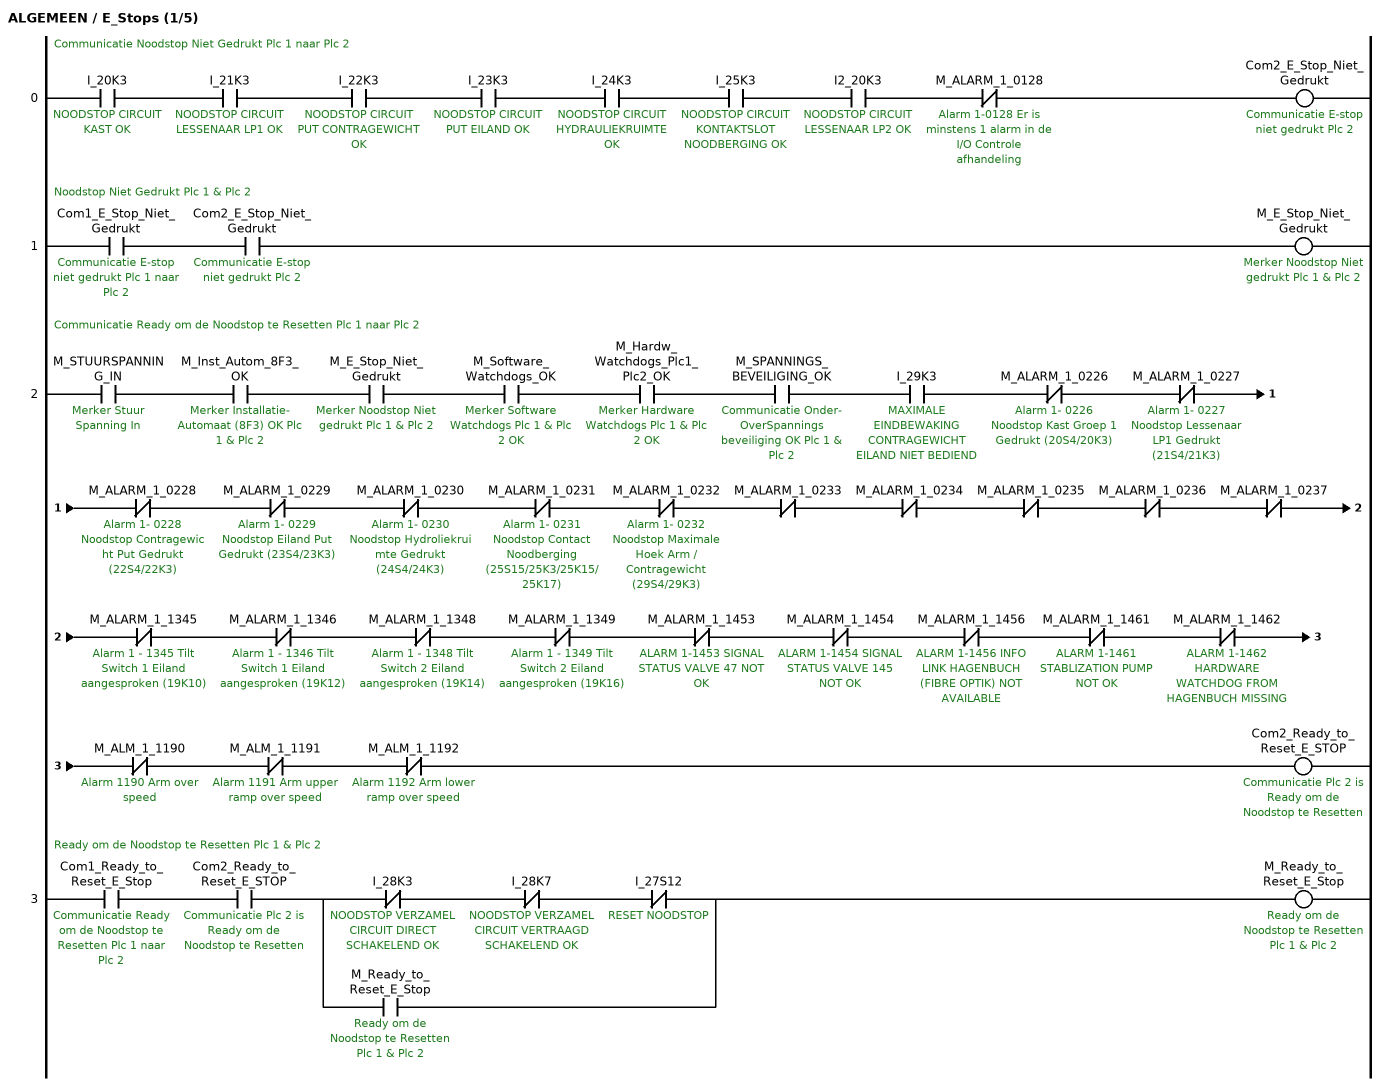
; rung 0: Communicatie Noodstop Niet Gedrukt Plc 1 naar Plc 2
LD I_20K3  ; NOODSTOP CIRCUIT KAST OK
AND I_21K3  ; NOODSTOP CIRCUIT LESSENAAR LP1 OK
AND I_22K3  ; NOODSTOP CIRCUIT PUT CONTRAGEWICHT OK
AND I_23K3  ; NOODSTOP CIRCUIT PUT EILAND OK
AND I_24K3  ; NOODSTOP CIRCUIT HYDRAULIEKRUIMTE OK
AND I_25K3  ; NOODSTOP CIRCUIT KONTAKTSLOT NOODBERGING OK
AND I2_20K3  ; NOODSTOP CIRCUIT LESSENAAR LP2 OK
ANDNOT M_ALARM_1_0128  ; Alarm 1-0128 Er is minstens 1 alarm in de I/O Controle afhandeling
OUT Com2_E_Stop_Niet_Gedrukt  ; Communicatie E-stop niet gedrukt Plc 2
; rung 1: Noodstop Niet Gedrukt Plc 1 & Plc 2
LD Com1_E_Stop_Niet_Gedrukt  ; Communicatie E-stop niet gedrukt Plc 1 naar Plc 2
AND Com2_E_Stop_Niet_Gedrukt  ; Communicatie E-stop niet gedrukt Plc 2
OUT M_E_Stop_Niet_Gedrukt  ; Merker Noodstop Niet gedrukt Plc 1 & Plc 2
; rung 2: Communicatie Ready om de Noodstop te Resetten Plc 1 naar Plc 2
LD M_STUURSPANNING_IN  ; Merker Stuur Spanning In
AND M_Inst_Autom_8F3_OK  ; Merker Installatie-Automaat (8F3) OK Plc 1 & Plc 2
AND M_E_Stop_Niet_Gedrukt  ; Merker Noodstop Niet gedrukt Plc 1 & Plc 2
AND M_Software_Watchdogs_OK  ; Merker Software Watchdogs Plc 1 & Plc 2 OK
AND M_Hardw_Watchdogs_Plc1_Plc2_OK  ; Merker Hardware Watchdogs Plc 1 & Plc 2 OK
AND M_SPANNINGS_BEVEILIGING_OK  ; Communicatie Onder- OverSpannings beveiliging OK Plc 1 & Plc 2
AND I_29K3  ; MAXIMALE EINDBEWAKING CONTRAGEWICHT EILAND NIET BEDIEND
ANDNOT M_ALARM_1_0226  ; Alarm 1- 0226 Noodstop Kast Groep 1 Gedrukt (20S4/20K3)
ANDNOT M_ALARM_1_0227  ; Alarm 1- 0227 Noodstop Lessenaar LP1 Gedrukt (21S4/21K3)
ANDNOT M_ALARM_1_0228  ; Alarm 1- 0228 Noodstop Contragewicht Put Gedrukt (22S4/22K3)
ANDNOT M_ALARM_1_0229  ; Alarm 1- 0229 Noodstop Eiland Put Gedrukt (23S4/23K3)
ANDNOT M_ALARM_1_0230  ; Alarm 1- 0230 Noodstop Hydroliekruimte Gedrukt (24S4/24K3)
ANDNOT M_ALARM_1_0231  ; Alarm 1- 0231 Noodstop Contact Noodberging (25S15/25K3/25K15/25K17)
ANDNOT M_ALARM_1_0232  ; Alarm 1- 0232 Noodstop Maximale Hoek Arm / Contragewicht  (29S4/29K3)
ANDNOT M_ALARM_1_0233
ANDNOT M_ALARM_1_0234
ANDNOT M_ALARM_1_0235
ANDNOT M_ALARM_1_0236
ANDNOT M_ALARM_1_0237
ANDNOT M_ALARM_1_1345  ; Alarm 1 - 1345 Tilt Switch 1 Eiland aangesproken (19K10)
ANDNOT M_ALARM_1_1346  ; Alarm 1 - 1346 Tilt Switch 1 Eiland aangesproken (19K12)
ANDNOT M_ALARM_1_1348  ; Alarm 1 - 1348 Tilt Switch 2 Eiland aangesproken (19K14)
ANDNOT M_ALARM_1_1349  ; Alarm 1 - 1349 Tilt Switch 2 Eiland aangesproken (19K16)
ANDNOT M_ALARM_1_1453  ; ALARM 1-1453 SIGNAL STATUS VALVE 47 NOT OK
ANDNOT M_ALARM_1_1454  ; ALARM 1-1454 SIGNAL STATUS VALVE 145 NOT OK
ANDNOT M_ALARM_1_1456  ; ALARM 1-1456 INFO LINK HAGENBUCH (FIBRE OPTIK) NOT AVAILABLE
ANDNOT M_ALARM_1_1461  ; ALARM 1-1461 STABLIZATION PUMP NOT OK
ANDNOT M_ALARM_1_1462  ; ALARM 1-1462 HARDWARE WATCHDOG FROM HAGENBUCH MISSING
ANDNOT M_ALM_1_1190  ; Alarm 1190 Arm over speed
ANDNOT M_ALM_1_1191  ; Alarm 1191 Arm upper ramp over speed
ANDNOT M_ALM_1_1192  ; Alarm 1192 Arm lower ramp over speed
OUT Com2_Ready_to_Reset_E_STOP  ; Communicatie Plc 2 is Ready om de Noodstop te Resetten
; rung 3: Ready om de Noodstop te Resetten Plc 1 & Plc 2
LD Com1_Ready_to_Reset_E_Stop  ; Communicatie Ready om de Noodstop te Resetten Plc 1 naar Plc 2
AND Com2_Ready_to_Reset_E_STOP  ; Communicatie Plc 2 is Ready om de Noodstop te Resetten
LDNOT I_28K3  ; NOODSTOP VERZAMEL CIRCUIT DIRECT SCHAKELEND OK
ANDNOT I_28K7  ; NOODSTOP VERZAMEL CIRCUIT VERTRAAGD SCHAKELEND OK
ANDNOT I_27S12  ; RESET NOODSTOP
OR M_Ready_to_Reset_E_Stop  ; Ready om de Noodstop te Resetten Plc 1 & Plc 2
ANDLD
OUT M_Ready_to_Reset_E_Stop  ; Ready om de Noodstop te Resetten Plc 1 & Plc 2

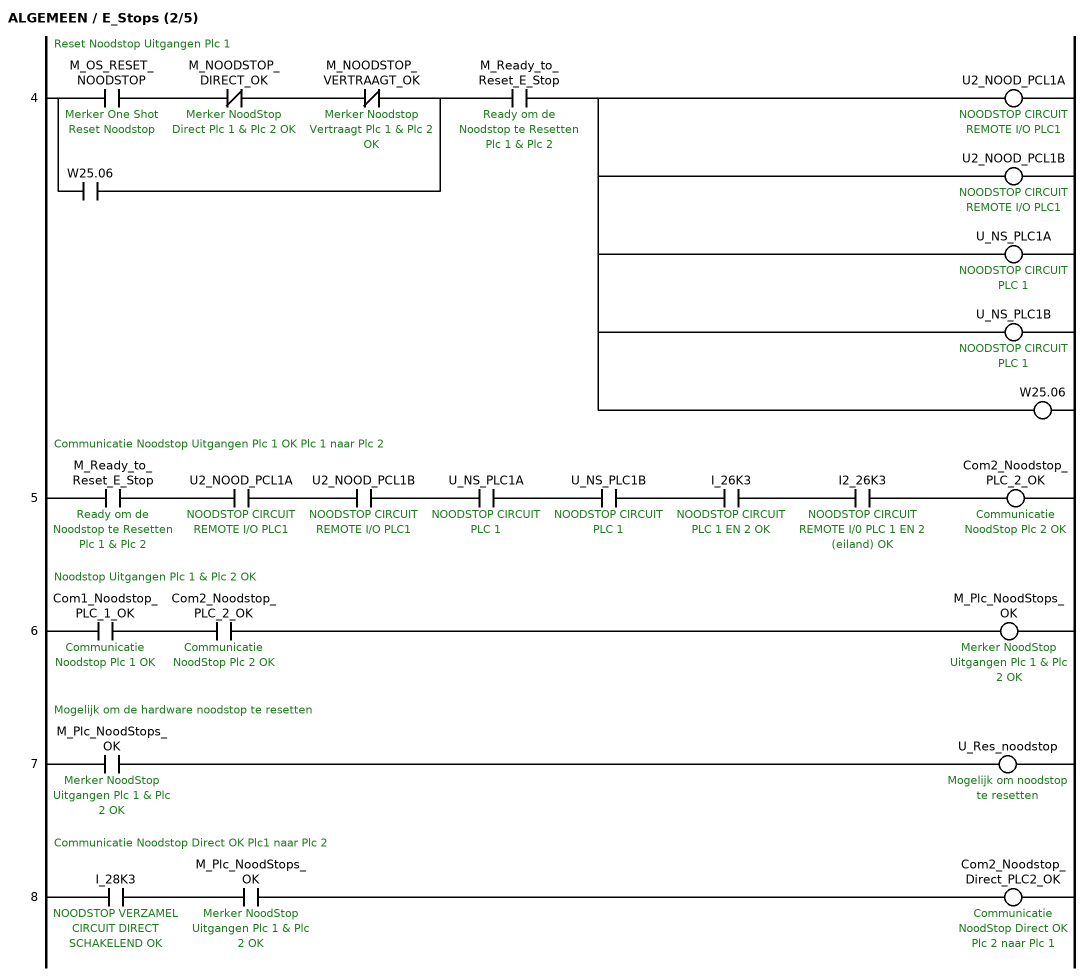
; rung 4: Reset Noodstop Uitgangen Plc 1
LD M_OS_RESET_NOODSTOP  ; Merker One Shot  Reset Noodstop
ANDNOT M_NOODSTOP_DIRECT_OK  ; Merker NoodStop Direct Plc 1 & Plc 2 OK
ANDNOT M_NOODSTOP_VERTRAAGT_OK  ; Merker Noodstop Vertraagt Plc 1 & Plc 2 OK
OR W25.06
AND M_Ready_to_Reset_E_Stop  ; Ready om de Noodstop te Resetten Plc 1 & Plc 2
OUT U2_NOOD_PCL1A  ; NOODSTOP CIRCUIT REMOTE I/O PLC1
OUT U2_NOOD_PCL1B  ; NOODSTOP CIRCUIT REMOTE I/O PLC1
OUT U_NS_PLC1A  ; NOODSTOP CIRCUIT PLC 1
OUT U_NS_PLC1B  ; NOODSTOP CIRCUIT PLC 1
OUT W25.06
; rung 5: Communicatie Noodstop Uitgangen Plc 1 OK Plc 1 naar Plc 2
LD M_Ready_to_Reset_E_Stop  ; Ready om de Noodstop te Resetten Plc 1 & Plc 2
AND U2_NOOD_PCL1A  ; NOODSTOP CIRCUIT REMOTE I/O PLC1
AND U2_NOOD_PCL1B  ; NOODSTOP CIRCUIT REMOTE I/O PLC1
AND U_NS_PLC1A  ; NOODSTOP CIRCUIT PLC 1
AND U_NS_PLC1B  ; NOODSTOP CIRCUIT PLC 1
AND I_26K3  ; NOODSTOP CIRCUIT PLC 1 EN 2 OK
AND I2_26K3  ; NOODSTOP CIRCUIT REMOTE I/0 PLC 1 EN 2 (eiland) OK
OUT Com2_Noodstop_PLC_2_OK  ; Communicatie NoodStop Plc 2 OK
; rung 6: Noodstop Uitgangen Plc 1 & Plc 2 OK
LD Com1_Noodstop_PLC_1_OK  ; Communicatie Noodstop Plc 1 OK
AND Com2_Noodstop_PLC_2_OK  ; Communicatie NoodStop Plc 2 OK
OUT M_Plc_NoodStops_OK  ; Merker NoodStop Uitgangen Plc 1 & Plc 2 OK
; rung 7: Mogelijk om de hardware noodstop te resetten
LD M_Plc_NoodStops_OK  ; Merker NoodStop Uitgangen Plc 1 & Plc 2 OK
OUT U_Res_noodstop  ; Mogelijk om noodstop te resetten
; rung 8: Communicatie Noodstop Direct OK Plc1 naar Plc 2
LD I_28K3  ; NOODSTOP VERZAMEL CIRCUIT DIRECT SCHAKELEND OK
AND M_Plc_NoodStops_OK  ; Merker NoodStop Uitgangen Plc 1 & Plc 2 OK
OUT Com2_Noodstop_Direct_PLC2_OK  ; Communicatie NoodStop Direct OK Plc 2 naar Plc 1

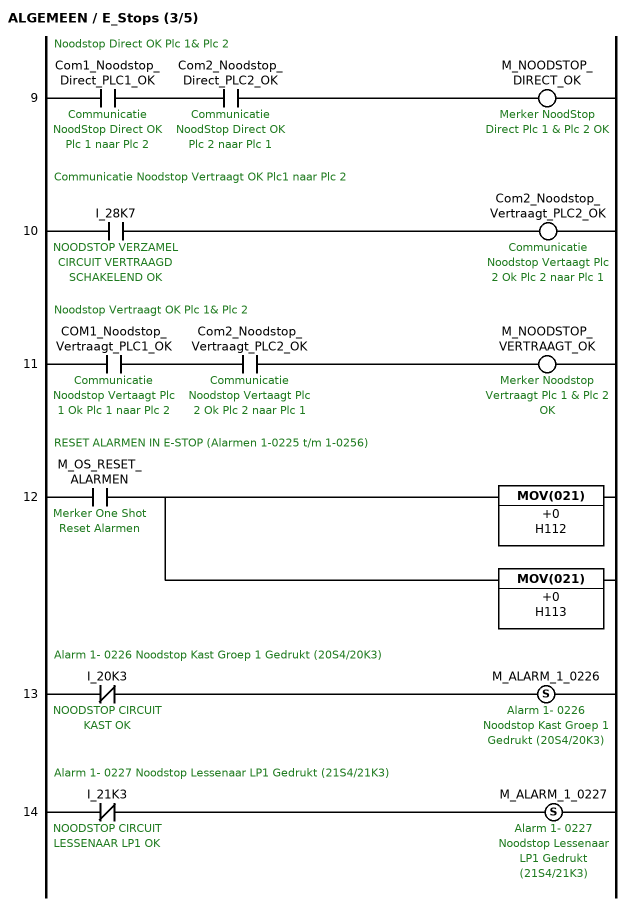
; rung 9: Noodstop Direct OK Plc 1& Plc 2
LD Com1_Noodstop_Direct_PLC1_OK  ; Communicatie NoodStop Direct OK Plc 1 naar Plc 2
AND Com2_Noodstop_Direct_PLC2_OK  ; Communicatie NoodStop Direct OK Plc 2 naar Plc 1
OUT M_NOODSTOP_DIRECT_OK  ; Merker NoodStop Direct Plc 1 & Plc 2 OK
; rung 10: Communicatie Noodstop Vertraagt OK Plc1 naar Plc 2
LD I_28K7  ; NOODSTOP VERZAMEL CIRCUIT VERTRAAGD SCHAKELEND OK
OUT Com2_Noodstop_Vertraagt_PLC2_OK  ; Communicatie Noodstop Vertaagt Plc 2 Ok Plc 2 naar Plc 1
; rung 11: Noodstop Vertraagt OK Plc 1& Plc 2
LD COM1_Noodstop_Vertraagt_PLC1_OK  ; Communicatie Noodstop Vertaagt Plc 1 Ok Plc 1 naar Plc 2
AND Com2_Noodstop_Vertraagt_PLC2_OK  ; Communicatie Noodstop Vertaagt Plc 2 Ok Plc 2 naar Plc 1
OUT M_NOODSTOP_VERTRAAGT_OK  ; Merker Noodstop Vertraagt Plc 1 & Plc 2 OK
; rung 12: RESET ALARMEN IN E-STOP (Alarmen 1-0225 t/m 1-0256)
LD M_OS_RESET_ALARMEN  ; Merker One Shot Reset Alarmen
MOV(021) +0 H112
MOV(021) +0 H113
; rung 13: Alarm 1- 0226 Noodstop Kast Groep 1 Gedrukt (20S4/20K3)
LDNOT I_20K3  ; NOODSTOP CIRCUIT KAST OK
SET M_ALARM_1_0226  ; Alarm 1- 0226 Noodstop Kast Groep 1 Gedrukt (20S4/20K3)
; rung 14: Alarm 1- 0227 Noodstop Lessenaar LP1 Gedrukt (21S4/21K3)
LDNOT I_21K3  ; NOODSTOP CIRCUIT LESSENAAR LP1 OK
SET M_ALARM_1_0227  ; Alarm 1- 0227 Noodstop Lessenaar LP1 Gedrukt (21S4/21K3)

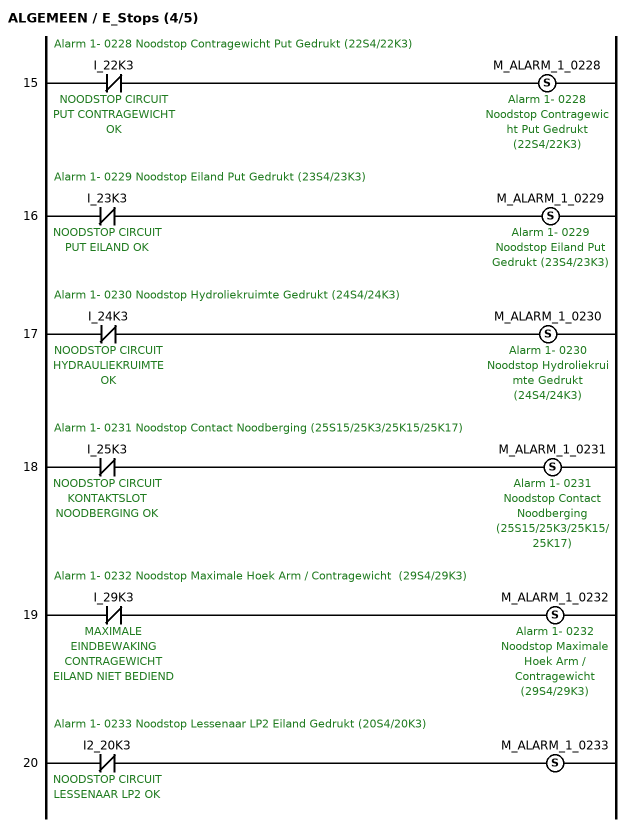
; rung 15: Alarm 1- 0228 Noodstop Contragewicht Put Gedrukt (22S4/22K3)
LDNOT I_22K3  ; NOODSTOP CIRCUIT PUT CONTRAGEWICHT OK
SET M_ALARM_1_0228  ; Alarm 1- 0228 Noodstop Contragewicht Put Gedrukt (22S4/22K3)
; rung 16: Alarm 1- 0229 Noodstop Eiland Put Gedrukt (23S4/23K3)
LDNOT I_23K3  ; NOODSTOP CIRCUIT PUT EILAND OK
SET M_ALARM_1_0229  ; Alarm 1- 0229 Noodstop Eiland Put Gedrukt (23S4/23K3)
; rung 17: Alarm 1- 0230 Noodstop Hydroliekruimte Gedrukt (24S4/24K3)
LDNOT I_24K3  ; NOODSTOP CIRCUIT HYDRAULIEKRUIMTE OK
SET M_ALARM_1_0230  ; Alarm 1- 0230 Noodstop Hydroliekruimte Gedrukt (24S4/24K3)
; rung 18: Alarm 1- 0231 Noodstop Contact Noodberging (25S15/25K3/25K15/25K17)
LDNOT I_25K3  ; NOODSTOP CIRCUIT KONTAKTSLOT NOODBERGING OK
SET M_ALARM_1_0231  ; Alarm 1- 0231 Noodstop Contact Noodberging (25S15/25K3/25K15/25K17)
; rung 19: Alarm 1- 0232 Noodstop Maximale Hoek Arm / Contragewicht  (29S4/29K3)
LDNOT I_29K3  ; MAXIMALE EINDBEWAKING CONTRAGEWICHT EILAND NIET BEDIEND
SET M_ALARM_1_0232  ; Alarm 1- 0232 Noodstop Maximale Hoek Arm / Contragewicht  (29S4/29K3)
; rung 20: Alarm 1- 0233 Noodstop Lessenaar LP2 Eiland Gedrukt (20S4/20K3)
LDNOT I2_20K3  ; NOODSTOP CIRCUIT LESSENAAR LP2 OK
SET M_ALARM_1_0233

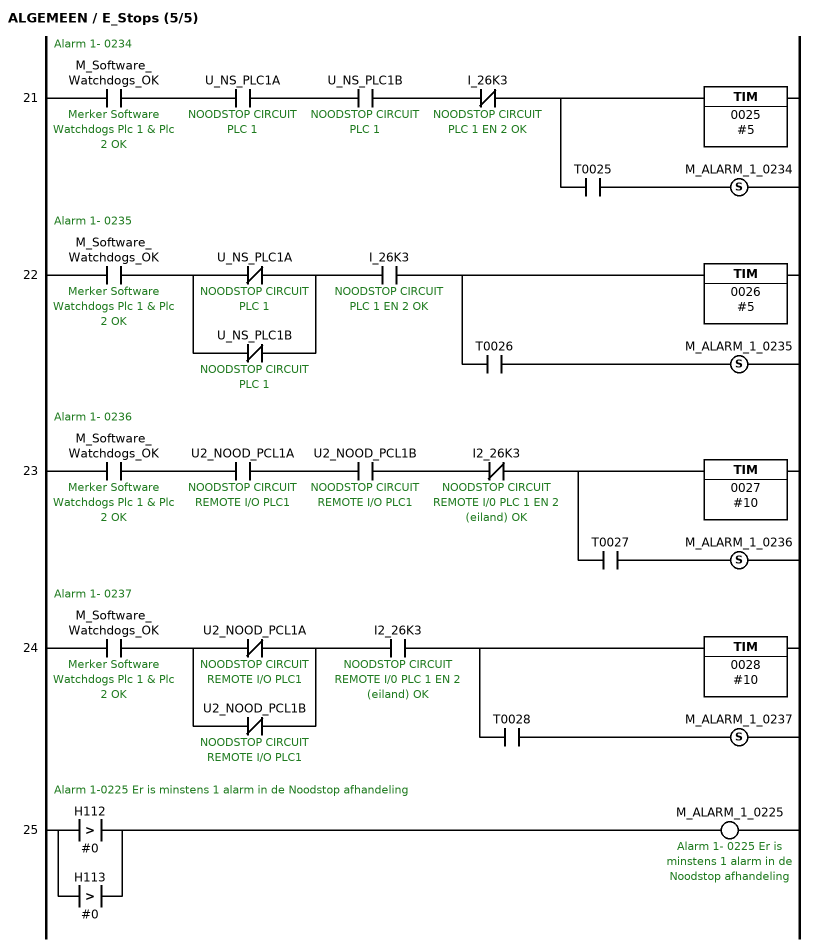
; rung 21: Alarm 1- 0234
LD M_Software_Watchdogs_OK  ; Merker Software Watchdogs Plc 1 & Plc 2 OK
AND U_NS_PLC1A  ; NOODSTOP CIRCUIT PLC 1
AND U_NS_PLC1B  ; NOODSTOP CIRCUIT PLC 1
ANDNOT I_26K3  ; NOODSTOP CIRCUIT PLC 1 EN 2 OK
TIM 0025 #5
AND T0025
SET M_ALARM_1_0234
; rung 22: Alarm 1- 0235
LD M_Software_Watchdogs_OK  ; Merker Software Watchdogs Plc 1 & Plc 2 OK
LDNOT U_NS_PLC1A  ; NOODSTOP CIRCUIT PLC 1
ORNOT U_NS_PLC1B  ; NOODSTOP CIRCUIT PLC 1
ANDLD
AND I_26K3  ; NOODSTOP CIRCUIT PLC 1 EN 2 OK
TIM 0026 #5
AND T0026
SET M_ALARM_1_0235
; rung 23: Alarm 1- 0236
LD M_Software_Watchdogs_OK  ; Merker Software Watchdogs Plc 1 & Plc 2 OK
AND U2_NOOD_PCL1A  ; NOODSTOP CIRCUIT REMOTE I/O PLC1
AND U2_NOOD_PCL1B  ; NOODSTOP CIRCUIT REMOTE I/O PLC1
ANDNOT I2_26K3  ; NOODSTOP CIRCUIT REMOTE I/0 PLC 1 EN 2 (eiland) OK
TIM 0027 #10
AND T0027
SET M_ALARM_1_0236
; rung 24: Alarm 1- 0237
LD M_Software_Watchdogs_OK  ; Merker Software Watchdogs Plc 1 & Plc 2 OK
LDNOT U2_NOOD_PCL1A  ; NOODSTOP CIRCUIT REMOTE I/O PLC1
ORNOT U2_NOOD_PCL1B  ; NOODSTOP CIRCUIT REMOTE I/O PLC1
ANDLD
AND I2_26K3  ; NOODSTOP CIRCUIT REMOTE I/0 PLC 1 EN 2 (eiland) OK
TIM 0028 #10
AND T0028
SET M_ALARM_1_0237
; rung 25: Alarm 1-0225 Er is minstens 1 alarm in de Noodstop afhandeling
LD>(320) H112 #0
OR>(320) H113 #0
OUT M_ALARM_1_0225  ; Alarm 1- 0225 Er is minstens 1 alarm in de Noodstop afhandeling

### Section Configure_I_O

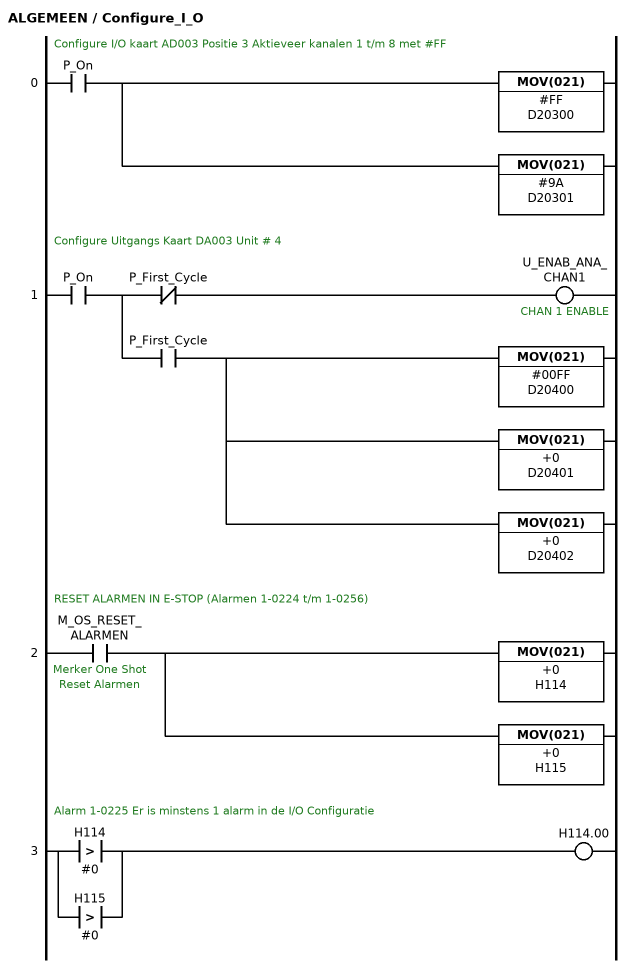
; rung 0: Configure I/O kaart AD003 Positie 3 Aktieveer kanalen 1 t/m 8 met #FF
LD P_On
MOV(021) #FF D20300
MOV(021) #9A D20301
; rung 1: Configure Uitgangs Kaart DA003 Unit # 4
LD P_On
OUT TR0
ANDNOT P_First_Cycle
OUT U_ENAB_ANA_CHAN1  ; CHAN 1 ENABLE
LD TR0
AND P_First_Cycle
MOV(021) #00FF D20400
MOV(021) +0 D20401
MOV(021) +0 D20402
; rung 2: RESET ALARMEN IN E-STOP (Alarmen 1-0224 t/m 1-0256)
LD M_OS_RESET_ALARMEN  ; Merker One Shot Reset Alarmen
MOV(021) +0 H114
MOV(021) +0 H115
; rung 3: Alarm 1-0225 Er is minstens 1 alarm in de I/O Configuratie
LD>(320) H114 #0
OR>(320) H115 #0
OUT H114.00

### Section Wind_Meting

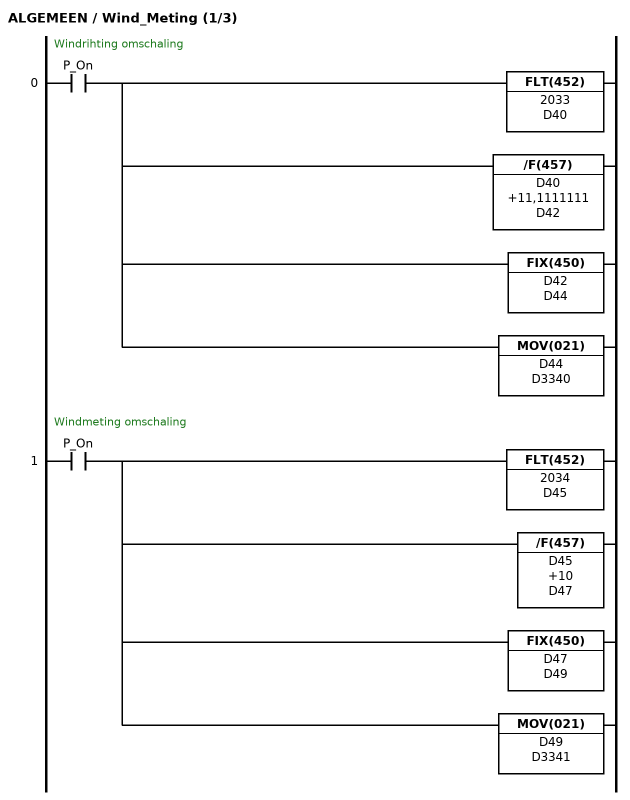
; rung 0: Windrihting omschaling
LD P_On
FLT(452) 2033 D40
/F(457) D40 +11,1111111 D42
FIX(450) D42 D44
MOV(021) D44 D3340
; rung 1: Windmeting omschaling
LD P_On
FLT(452) 2034 D45
/F(457) D45 +10 D47
FIX(450) D47 D49
MOV(021) D49 D3341

